PROGRAM Analog_IO_Mapping
VAR
END_VAR

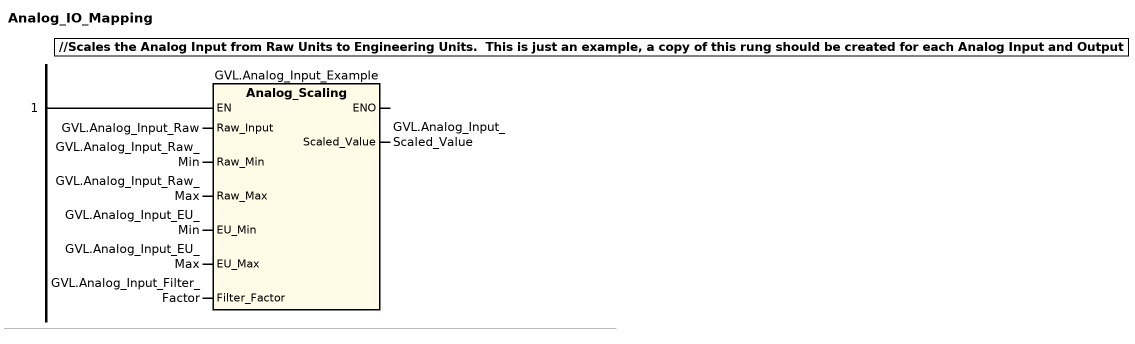
// NETWORK 1
// label: //Scales the Analog Input from Raw Units to Engineering Units.  This is just an example, a copy of this rung should be created for each Analog Input and Output
GVL.Analog_Input_Example(
    Raw_Input := GVL.Analog_Input_Raw,
    Raw_Min := GVL.Analog_Input_Raw_Min,
    Raw_Max := GVL.Analog_Input_Raw_Max,
    EU_Min := GVL.Analog_Input_EU_Min,
    EU_Max := GVL.Analog_Input_EU_Max,
    Filter_Factor := GVL.Analog_Input_Filter_Factor,
    Scaled_Value => GVL.Analog_Input_Scaled_Value); // Analog_Scaling

END_PROGRAM

(* stored: Version 1.1.0.1, ProductVersion 3.1.4024.12
   POU Analog_IO_Mapping: Id {9d147058-5126-4261-979a-bdb9d4f76c05}, SpecialFunc None *)
